FUNCTION TryConvert_TOD_TO_USINT : BOOL
VAR_INPUT
	in : TOD;
	out : REFERENCE TO USINT;
END_VAR

IF in > DatatypeLimits.MAX_VALUE_OF_TOD_WHICH_CAN_BE_HELD_IN_A_USINT THEN
	RETURN;
END_IF

out := TOD_TO_USINT(in);
TryConvert_TOD_TO_USINT := TRUE;

END_FUNCTION

(* stored: Version 1.1.0.1, ProductVersion 3.1.4024.12
   POU TryConvert_TOD_TO_USINT: Id {8399c67f-d1b9-4612-aeca-c730cbea6ddb}, SpecialFunc None *)
